ABB RobotStudio station: Tp1.rsstn

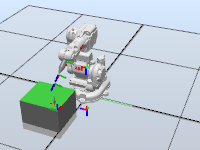
Station Tp1 (saved by RobotStudio 20.2.9116.0)
Controller IRB_140_6kg_0.81m
  mechanical unit ROB_1: IRB140_6_81_C_03, 6 joints, base frame (0, 0, 0) mm
Layout (positions relative to the parent item):
  - IRB140_6_81_C_03 [mechanism, from Robots\IRB140_6_81_C_G_03.rslib] at (0, 0, 0) mm; joint values [0, -0.0689, 0.0956, 0, 0.4969, 0] (rad or m)
  - Mesa [part]
  - Perno [part] at (200, 70, 180) mm, rotated rx 90 ry 0 rz 0 deg
  - Pinza [mechanism] at (481.35, 0, 668.5) mm, rotated rx -180 ry 60 rz -180 deg
      TCP Pinza at (0, 0, 137) mm, rotated rx 0 ry 0 rz -22.5 deg
      links: Dummy
Attachment: Pinza is attached to IRB140_6_81_C_03 / Link6
EventTableEntry 1017: Group=, Trigger=DO_Pinza 1018, Actions=[EventTableActionAttach 1019], Comment=, ActivationMode=2, Cyclic=false
EventTableTriggerIO 1018: IOValue=[1], IRC5Controller=? -1, Operator=0, SignalSource=IRB_140_6kg_0.81m 515
EventTableActionAttach 1019: AttachmentParent=Pinza 1013, AttachmentChild=Perno 1009, MountObject=false, Offset=[X=1, Y=0, Z=0, W=0, X=0, Y=1, Z=0, W=0, X=0, Y=0, Z=1, W=0, X=0, Y=0, Z=0, W=1], FlangeIndext=0, FindNearest=false
EventTableEntry 1020: Group=, Trigger=DO_Pinza 1021, Actions=[EventTableActionDetach 1022], Comment=, ActivationMode=2, Cyclic=false
EventTableTriggerIO 1021: IOValue=[0], IRC5Controller=? -1, Operator=0, SignalSource=IRB_140_6kg_0.81m 515
EventTableActionDetach 1022: AttachmentParent=Pinza 1013, AttachmentChild=Perno 1009
Collision set Colision Perno- Mesa: Perno against Mesa, near miss 0.0009 m
Collision set Colision Robot - Mesa: IRB140_6_81_C_03 against Mesa, near miss 0 m
Collision set Colision Pinza - Mesa: Mesa against Pinza, near miss 0 m
EventTableTriggerIO 1093: IOValue=[1], IRC5Controller=? -1, Operator=0, SignalSource=IRB_140_6kg_0.81m 515
EventTableTriggerIO 1094: IOValue=[0], IRC5Controller=? -1, Operator=0, SignalSource=IRB_140_6kg_0.81m 515
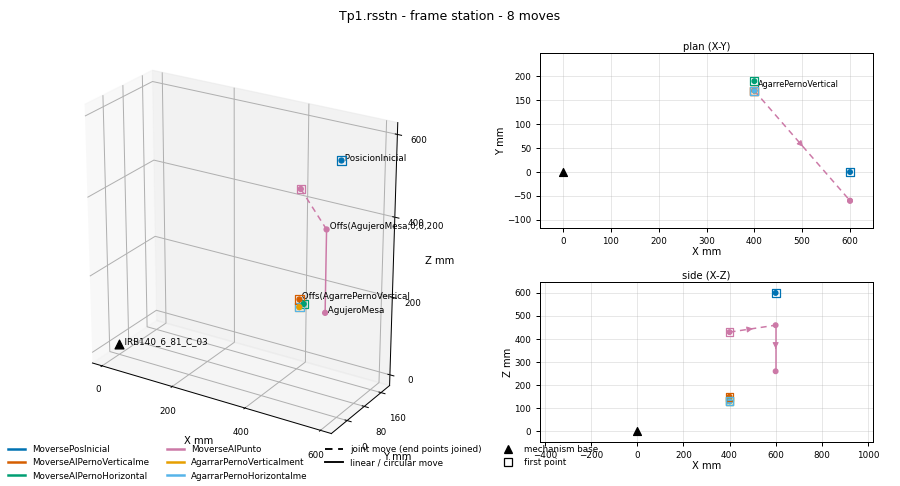
[picture p0: tool path of Tp1.rsstn in frame station, 8 of 12 moves have a stored position in this frame; points joined in program order, loops and branches not executed]
Targets, tools, work objects and paths stored in the station, written as RAPID:
! task T_ROB1
MODULE Module1
  PERS tooldata Pinza:=[TRUE,[[0,0,137],[0.980785,0,0,-0.19509]],[0.5,[0,0,100],[1,0,0,0],0,0,0]];
  PERS wobjdata wobjMesa:=[FALSE,TRUE,"",[[665,5,260],[0,0,0,1]],[[0,0,0],[1,0,0,0]]];
  CONST robtarget PosicionInicial:=[[600,0,600],[0.490392593,-0.168953224,0.849384987,-0.097545151],[-1,0,-1,0],[9E+09,9E+09,9E+09,9E+09,9E+09,9E+09]];
  CONST robtarget AgujeroMesa:=[[65,65,0],[0,0.707106781,0.707106781,0],[-1,0,-2,0],[9E+09,9E+09,9E+09,9E+09,9E+09,9E+09]];
  CONST robtarget AgarrePernoVertical:=[[400,170,130],[0,-0.707106781,0.707106781,0],[0,0,-1,0],[9E+09,9E+09,9E+09,9E+09,9E+09,9E+09]];
  CONST robtarget ReorientacionVertical:=[[400.000008995,170.000009452,600.000002468],[-0.000000008,0.707106992,-0.707106571,0.000000082],[0,1,1,1],[9E+09,9E+09,9E+09,9E+09,9E+09,9E+09]];
  CONST robtarget AgarrePernoHorizontal:=[[400,170,130],[0.5,0.5,-0.5,0.5],[0,-1,0,0],[9E+09,9E+09,9E+09,9E+09,9E+09,9E+09]];
  PERS tooldata Pinza_Perno:=[TRUE,[[0,0,227],[0.980785,0,0,-0.19509]],[0.1,[0,0,100],[1,0,0,0],0,0,0]];
  PROC main()
    MoversePosInicial;
    MoverseAlPernoHorizontalmente;
    AgarrarPernoHorizontalmente;
    MoverseAlPernoVerticalmente;
    AgarrarPernoVerticalmente;
    EnviarMensajeError;
    MoverseAlPunto;
    SoltarPerno;
    MoversePosInicial;
  ENDPROC
  PROC MoversePosInicial()
    MoveJ PosicionInicial,Velocidad,fine,Pinza\WObj:=wobj0;
  ENDPROC
  PROC MoverseAlPernoVerticalmente()
    MoveL aux,Velocidad,fine,Pinza\WObj:=wobj0;
    MoveL aux,Velocidad,fine,Pinza\WObj:=wobj0;
    MoveJ Offs(AgarrePernoVertical,0,0,20),Velocidad,fine,Pinza\WObj:=wobj0;
  ENDPROC
  PROC MoverseAlPernoHorizontalmente()
    MoveL aux,Velocidad,fine,Pinza\WObj:=wobj0;
    MoveL aux,Velocidad,fine,Pinza\WObj:=wobj0;
    MoveJ Offs(AgarrePernoHorizontal,0,20,0),Velocidad,fine,Pinza\WObj:=wobj0;
  ENDPROC
  PROC AgarrarPerno()
    SetDO DO_Pinza,1;
  ENDPROC
  PROC SoltarPerno()
    SetDO DO_Pinza,0;
  ENDPROC
  PROC MoverseAlPunto()
    MoveL Offs(AgarrePernoVertical,0,0,300),Velocidad,fine,Pinza\WObj:=wobj0;
    ConfJ \On;
    MoveJ Offs(AgujeroMesa,0,0,200),Velocidad,fine,Pinza_Perno\WObj:=wobjMesa;
    MoveL AgujeroMesa,Velocidad,fine,Pinza_Perno\WObj:=wobjMesa;
  ENDPROC
  PROC EnviarMensajeError()
  ENDPROC
  PROC AgarrarPernoVerticalmente()
    MoveJ AgarrePernoVertical,Velocidad,fine,Pinza\WObj:=wobj0;
    SetDO DO_Pinza,1;
  ENDPROC
  PROC AgarrarPernoHorizontalmente()
    MoveJ AgarrePernoHorizontal,Velocidad,fine,Pinza\WObj:=wobj0;
    SetDO DO_Pinza,1;
  ENDPROC
ENDMODULE

